FUNCTION_BLOCK FB_GantryDifferenceMonitor
VAR_IN_OUT
	Gantry	:	HOMS_Gantry;
END_VAR
VAR_INPUT
END_VAR
VAR_OUTPUT
END_VAR
VAR
END_VAR
VAR CONSTANT
	
END_VAR

(* Gantry Difference Monitor
E. Rodriguez, A. Wallace 17-2-15

The gantry difference monitor runs in a fast task and monitors
the gantry difference between two gantried axes. If this difference
exceeds the permitted amount, a gauntry fault boolean is set. 

Axilon provided encoder counts for the "center" of each axis. We 
consider this center to be the zero-gantry-difference position.

This boolean is monitored by other function blocks that use the gantry structure, including
but not limited to:
Gantry control function block
System error summary
*)

//1 encoder count = 1 nm
//AxilonGantryDiff := Gantry.PAxis.cCenter - Gantry.SAxis.cCenter;

//HOMSGantryDiff := Gantry.PAxis.diEncCnt - Gantry.SAxis.diEncCnt;

Gantry.Diff := LREAL_TO_REAL(Gantry.PAxis.stAxis.NcToPlc.ActPos - Gantry.SAxis.stAxis.NcToPlc.ActPos);

Gantry.DiffFlt S= ABS(Gantry.Diff) > Gantry.DiffTol;
Gantry.DiffFlt R= ABS(Gantry.Diff) <= Gantry.DiffTol - Gantry.DiffHys;

END_FUNCTION_BLOCK

(* stored: Version 1.1.0.1, ProductVersion 3.1.4024.6
   POU FB_GantryDifferenceMonitor: Id {e176ae5e-8c7a-4621-9b04-821738e2daeb}, SpecialFunc None *)
